// Device/Application/Vizualization/7_inch/_Actuators
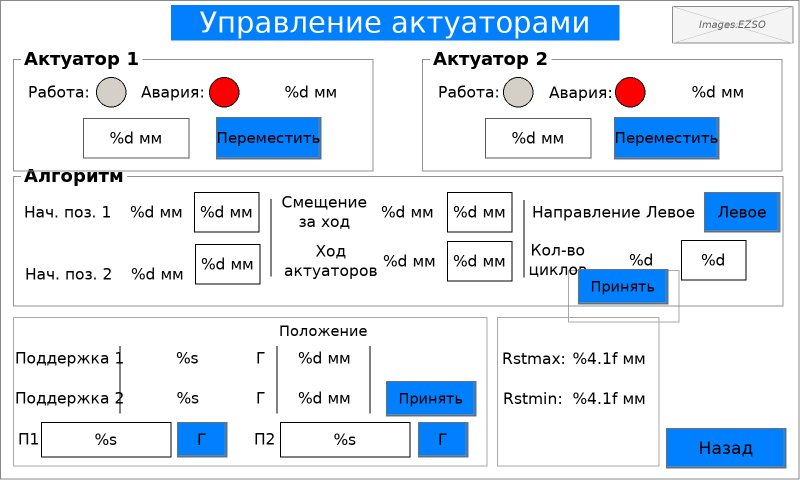
VISUALIZATION _Actuators  // 800x480, background image Images.background
    RoundedRectangle (568,270 111x52)
    GroupBox (13,168 770x138), "Алгоритм"
        Label (507,75 76x34), "Кол-во циклов"
        Label (516,27 113x34), "Направление"
        Button (691,24 76x40), "Левое", text list: 'DirectRotation', text index: setPoint.bDirRotate
            toggle setPoint.bDirRotate
        RoundedRectangle (668,72 65x40), "%d", text variable: setPoint.iCountCycle
            OnMouseClick: write the text variable via VisuDialogs.Numpad, min 0, max 360, title 'Input'
        RoundedRectangle (181,24 65x40), "%d мм", text variable: setPoint.iActuatorsStartPos[0]
            OnMouseClick: write the text variable via VisuDialogs.Numpad, min 0, max SP.iMaxActuatorsMove, title 'Input'
        RoundedRectangle (434,24 65x40), "%d мм", text variable: setPoint.iActuatorsStep
            OnMouseClick: write the text variable via VisuDialogs.Numpad, min 0, max SP.iMaxActuatorsMove, title 'Input'
        Label (8,27 98x34), "Нач. поз. 1"
        Label (260,27 103x34), "Смещение за ход"
        Rectangle (111,29 65x30), "%d мм", text variable: curPoint.iActuatorsStartPos[0]
        Line (258,108) (258,31)
        Line (511,109) (511,32)
        Rectangle (596,77 65x30), "%d", text variable: curPoint.iCountCycle
        Rectangle (362,29 65x30), "%d мм", text variable: curPoint.iActuatorsStep
        Rectangle (625,29 65x30), "Левое", text list: 'DirectRotation', text index: curPoint.bDirRotate
        Button (565,101 90x35), "Принять", pressed state: Global_Variables.btnAccept.bAct
            tap Global_Variables.btnAccept.bAct
        RoundedRectangle (182,76 65x40), "%d мм", text variable: setPoint.iActuatorsStartPos[1]
            OnMouseClick: write the text variable via VisuDialogs.Numpad, min 0, max SP.iMaxActuatorsMove, title 'Input'
        Rectangle (364,78 65x30), "%d мм", text variable: curPoint.iActuatorsMove
        RoundedRectangle (434,73 65x40), "%d мм", text variable: setPoint.iActuatorsMove
            OnMouseClick: write the text variable via VisuDialogs.Numpad, min 0, max SP.iMaxActuatorsMove, title 'Input'
        Label (271,76 94x34), "Ход актуаторов"
    RoundedRectangle (497,317 162x149)
    RoundedRectangle (13,317 474x149)
    Image (672,6 121x37), image: Images.EZSO
    Button (666,428 120x40), "Назад"
        OnMouseDown:  Assign=_MAIN_7inch, Type=Previous
        OnMouseDown: execute { Actuators.bManualMode := FALSE; }
    Rectangle (171,5 448x35), "Управление актуаторами"
    GroupBox (13,51 360x120), "Актуатор 1"
        RoundedRectangle (70,67 106x40), "%d мм", text variable: Actuators.fbAct1.iSetp
            OnMouseClick: write the text variable via VisuDialogs.Numpad, min 0, max SP.rMaxLength, title 'Input'
        Button (203,66 105x42), "Переместить", pressed state: Actuators.fbAct1.bBtnStart
            tap Actuators.fbAct1.bBtnStart
        Rectangle (240,26 116x30), "%d мм", text variable: Actuators.fbAct1.iCurLength
        Label (12,25 68x32), "Работа:"
        Ellipse (83,26 30x30), colour toggle: Actuators.bDr1_enable
        Label (125,25 68x32), "Авария:"
        Ellipse (196,26 30x30), colour toggle: Actuators.bDr2_error
    GroupBox (422,51 360x120), "Актуатор 2"
        RoundedRectangle (63,67 106x40), "%d мм", text variable: Actuators.fbAct2.iSetp
            OnMouseClick: write the text variable via VisuDialogs.Numpad, min 0, max SP.rMaxLength, title 'Input'
        Button (192,66 105x42), "Переместить", pressed state: Actuators.fbAct2.bBtnStart
            tap Actuators.fbAct2.bBtnStart
        Rectangle (238,26 116x30), "%d мм", text variable: Actuators.fbAct2.iCurLength
        Label (13,24 67x34), "Работа:"
        Ellipse (81,26 30x30), colour toggle: Actuators.bDr1_enable
        Label (124,26 68x31), "Авария:"
        Ellipse (193,26 30x30), colour toggle: Actuators.bDr2_error
    Line (120,413) (120,346)
    Line (277,413) (277,346)
    Button (418,422 50x35), "Г", text list: 'TypeSetup', text index: setPoint.support[1].bPosition
        toggle setPoint.support[1].bPosition
    Button (177,422 50x35), "Г", text list: 'TypeSetup', text index: setPoint.support[0].bPosition
        toggle setPoint.support[0].bPosition
    RoundedRectangle (280,422 130x35), "%s", text variable: setPoint.support[1].name
        OnMouseClick:  Dialog=_Diag_supKey, Parameters={stValue: setPoint.support[1]}, Selected={1: }, OpenModal=True, PositionX=300, PositionY=150
    RoundedRectangle (41,422 130x35), "%s", text variable: setPoint.support[0].name
        OnMouseClick:  Dialog=_Diag_supKey, Parameters={stValue: setPoint.support[0]}, Selected={1: }, OpenModal=True, PositionX=300, PositionY=150
    Label (12,381 105x34), "Поддержка 2"
    Label (12,341 105x34), "Поддержка 1"
    Line (370,413) (370,346)
    Label (276,314 96x34), "Положение"
    Rectangle (286,343 77x30), "%d мм", text variable: Actuators.iCurLenSuport1
    Rectangle (286,383 77x30), "%d мм", text variable: Actuators.iCurLenSuport2
    RoundedRectangle (564,341 90x35), "%4.1f мм", text variable: curPoint.rRstmax
    Label (499,343 66x31), "Rstmax:"
    Label (500,383 65x31), "Rstmin:"
    RoundedRectangle (564,381 90x35), "%4.1f мм", text variable: curPoint.rRstmin
    Rectangle (123,343 129x30), "%s", text variable: curPoint.support[0].name
    Rectangle (123,383 130x30), "%s", text variable: curPoint.support[1].name
    Rectangle (246,343 30x30), "Г", text list: 'TypeSetup', text index: curPoint.support[0].bPosition
    Rectangle (246,383 30x30), "Г", text list: 'TypeSetup', text index: curPoint.support[1].bPosition
    Button (386,381 90x35), "Принять", pressed state: Global_Variables.btnAccept.bSup
        tap Global_Variables.btnAccept.bSup
    Label (15,426 31x26), "П1"
    Label (251,426 31x26), "П2"
    Label (22,257 98x34), "Нач. поз. 2"
    Rectangle (125,259 65x30), "%d мм", text variable: curPoint.iActuatorsStartPos[1]
END_VISUALIZATION

// Device/Application/Vizualization/7_inch/_SettingsEquipment
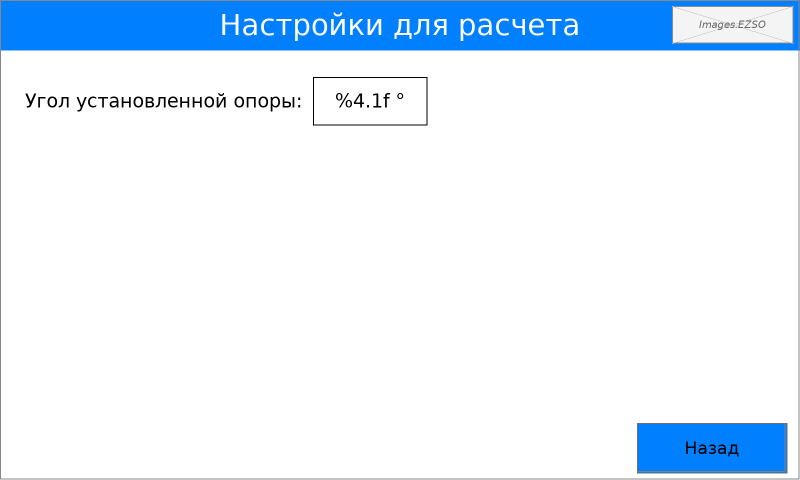
VISUALIZATION _SettingsEquipment  // 800x480
    Rectangle (0,0 800x50), "Настройки для расчета"
    Image (672,6 121x37), image: Images.EZSO
    Button (637,423 150x50), "Назад"
        OnMouseDown:  Assign=_MAIN_7inch, Type=Previous
    RoundedRectangle (313,77 114x48), "%4.1f °", text variable: SP.rInitAngleSupport
        OnValueChanged: execute { CalcTech.rAngle_support:=sp.rInitAngleSupport; }
        OnMouseClick: write the text variable via VisuDialogs.Numpad, min 0, max 359
    Label (22,80 295x42), "Угол установленной опоры:"
END_VISUALIZATION

// Device/Application/Vizualization/7_inch/_Diag_geomtry_rec
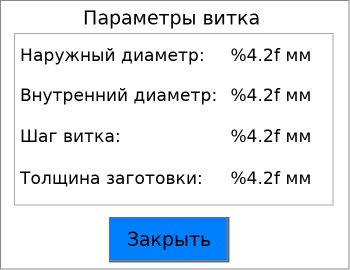
VISUALIZATION _Diag_geomtry_rec  // 350x270
    Button (109,217 120x45), "Закрыть"
        toggle bGoCalc
        OnMouseClick:  Dialog=Current Dialog, Result=OK, NumpadKeypadSet=True
    RoundedRectangle (214,71 114x48), "%4.2f мм", text variable: recipes.Screw.rInner_diam
    Label (17,74 223x42), "Внутренний диаметр:"
    RoundedRectangle (214,31 114x48), "%4.2f мм", text variable: recipes.Screw.rOut_diam
        OnMouseClick: write the text variable via VisuDialogs.Numpad
    Label (17,34 223x42), "Наружный диаметр:"
    RoundedRectangle (214,112 114x48), "%4.2f мм", text variable: recipes.Screw.rTurn_step
    Label (17,115 223x42), "Шаг витка:"
    RoundedRectangle (214,154 114x48), "%4.2f мм", text variable: recipes.Screw.rWidth
    Label (17,157 223x42), "Толщина заготовки:"
    Label (80,1 185x34), "Параметры витка"
    RoundedRectangle (14,33 319x172)
END_VISUALIZATION

// Device/Application/Vizualization/7_inch/_Support
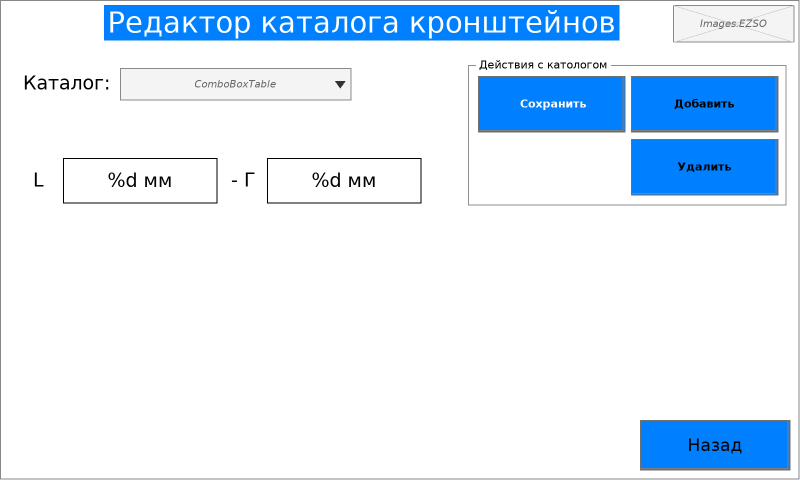
VISUALIZATION _Support  // 800x480, background image Images.background
    GroupBox (468,57 318x148), "Действия с катологом"
        Button (163,82 147x56), "Удалить"
            OnMouseClick: execute { recipes.DelData(3); }
        Button (163,19 147x56), "Добавить"
            OnMouseClick: execute { recipes.addData(3); }
        Button (10,19 147x56), "Сохранить"
            OnMouseClick: execute { recipes.setData(3); }
    Label (30,165 31x30), "L"
    Label (20,68 99x30), "Каталог:"
    Image (673,5 121x37), image: Images.EZSO
    Rectangle (104,5 515x35), "Редактор каталога кронштейнов"
    Button (640,420 150x50), "Назад"
        OnMouseDown:  Assign=_Equipment, Type=Assignment
        OnMouseDown:  ExecuteCommand=ExecuteCommand=[Command=ReadRecipe, Value=sRecGroupName3, Value2=sRecName3]
    ComboBoxTable (120,68 231x32), variable: recipes.idxArSupport, data array: arSupports
        p1014161805: Global_Variables.SIZE_SUPPORT - 0 + 1
        p338671338: arrSteel_buf[INDEX].G
        p2170511999: arrSteel_buf[INDEX].t
        p3854506369: arSupports[INDEX].arLength
        p1892666644: arSupports[INDEX].name
        OnValueChanged: execute { recipes.GetData(3); }
    RoundedRectangle (63,158 154x45), "%d мм", text variable: recipes.Support.arLength[0]
        OnMouseClick: write the text variable via VisuDialogs.Numpad, min -999, max 999, title 'Input'
    RoundedRectangle (267,158 154x45), "%d мм", text variable: recipes.Support.arLength[1]
        OnMouseClick: write the text variable via VisuDialogs.Numpad, min -999, max 999, title 'Input'
    Label (228,165 31x30), "- Г"
END_VISUALIZATION

// Device/Application/Vizualization/7_inch/_Equipment_2
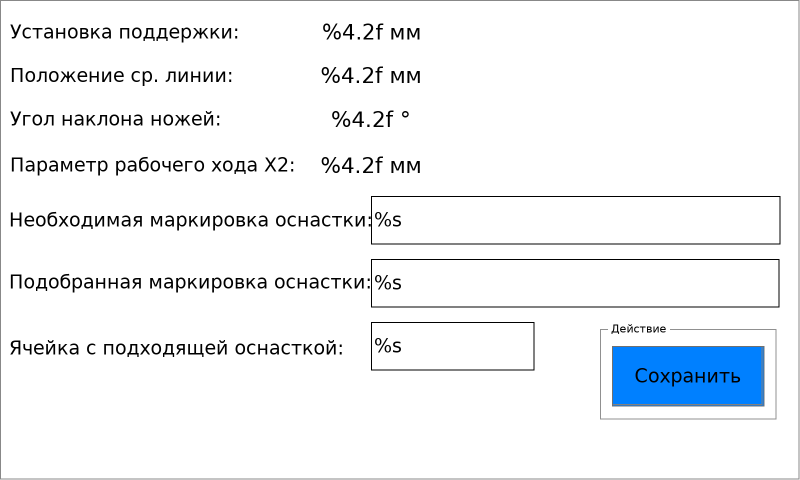
VISUALIZATION _Equipment_2  // 800x480
    Label (6,327 338x42), "Ячейка с подходящей оснасткой:"
    Label (6,198 396x44), "Необходимая маркировка оснастки:"
    RoundedRectangle (371,196 409x48), "%s", text variable: CalcTech.msEquipment.bestFind.name
    Label (7,55 231x41), "Положение ср. линии:"
    Label (7,15 232x34), "Установка поддержки:"
    RoundedRectangle (371,259 408x48), "%s", text variable: CalcTech.msEquipment.find.name
    Label (7,98 223x42), "Угол наклона ножей:"
    Label (7,144 322x42), "Параметр рабочего хода Х2:"
    Label (6,261 360x42), "Подобранная маркировка оснастки:"
    Rectangle (322,17 100x30), "%4.2f мм", text variable: CalcTech.rMsFactInstal_support
    Rectangle (320,62 102x27), "%4.2f мм", text variable: CalcTech.rMsFactMidle_line
    Rectangle (320,152 102x27), "%4.2f мм", text variable: CalcTech.rMsX2
    Rectangle (320,106 102x27), "%4.2f °", text variable: CalcTech.rMsAngle_knives
    RoundedRectangle (371,322 163x48), "%s", text variable: CalcTech.msEquipment.find.place
    GroupBox (600,321 176x98), "Действие"
        Button (12,25 152x60), "Сохранить"
            OnMouseClick:  Dialog=_Diag_save, PositionX=300, PositionY=150
END_VISUALIZATION

// Device/Application/Vizualization/7_inch/_Equipment_3
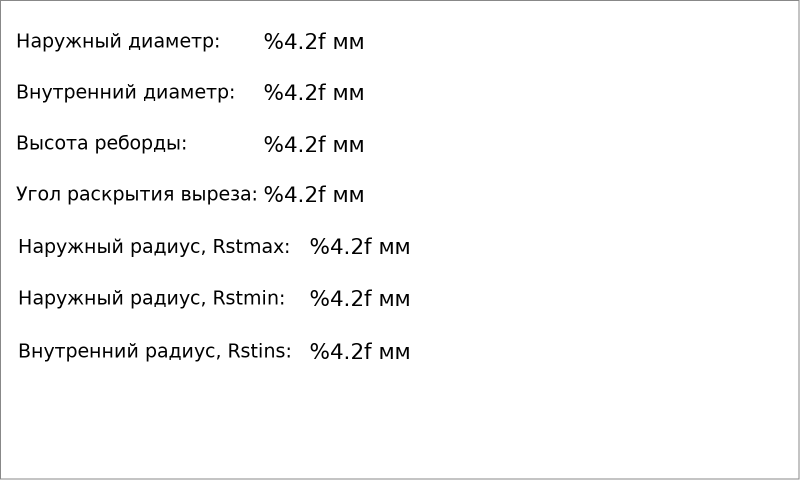
VISUALIZATION _Equipment_3  // 800x480
    Label (13,71 223x42), "Внутренний диаметр:"
    Label (13,20 223x42), "Наружный диаметр:"
    Label (13,122 223x42), "Высота реборды:"
    Label (13,173 250x42), "Угол раскрытия выреза:"
    Rectangle (263,181 102x27), "%4.2f мм", text variable: CalcTech.rWpAngle
    Rectangle (263,79 102x27), "%4.2f мм", text variable: CalcTech.rWpInner_diam
    Rectangle (263,28 102x27), "%4.2f мм", text variable: CalcTech.rWpOut_diam
    Rectangle (263,131 102x27), "%4.2f мм", text variable: CalcTech.rWpRebordHeight
    Label (15,224 290x45), "Наружный радиус, Rstmax:", invisible if: not CalcTech.bEnConicalScrew
    Rectangle (309,234 102x25), "%4.2f мм", text variable: CalcTech.rRstmax, invisible if: not CalcTech.bEnConicalScrew
    Label (15,278 290x40), "Наружный радиус, Rstmin:", invisible if: not CalcTech.bEnConicalScrew
    Label (15,331 289x40), "Внутренний радиус, Rstins:", invisible if: not CalcTech.bEnConicalScrew
    Rectangle (309,286 102x25), "%4.2f мм", text variable: CalcTech.rRstmin, invisible if: not CalcTech.bEnConicalScrew
    Rectangle (309,339 102x25), "%4.2f мм", text variable: CalcTech.rRstins, invisible if: not CalcTech.bEnConicalScrew
END_VISUALIZATION

// Device/Application/Vizualization/7_inch/_Diag_WARNING
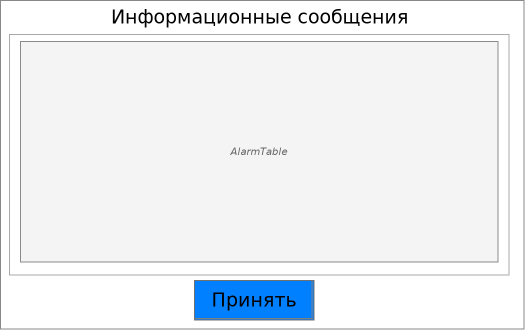
VISUALIZATION _Diag_WARNING  // 525x330
VAR_IN_OUT
	stValue:WSTRING;	
END_VAR
VAR
	sDirection: INT;
	sTypeEquip:	INT;
	sHeight: WSTRING;
	sAngle:	WSTRING;
	sMidle:	WSTRING;	
END_VAR
    RoundedRectangle (9,34 500x241)
    Button (194,280 120x40), "Принять"
        tap bReset
        OnMouseDown:  Dialog=Current Dialog, Result=OK, NumpadKeypadSet=True
    AlarmTable (20,41 478x221)
        p1521930926: WarningGroup
        p1663851261: Warning
    Label (108,0 308x34), "Информационные сообщения"
END_VISUALIZATION

// Device/Application/Vizualization/7_inch/_TypeMachine
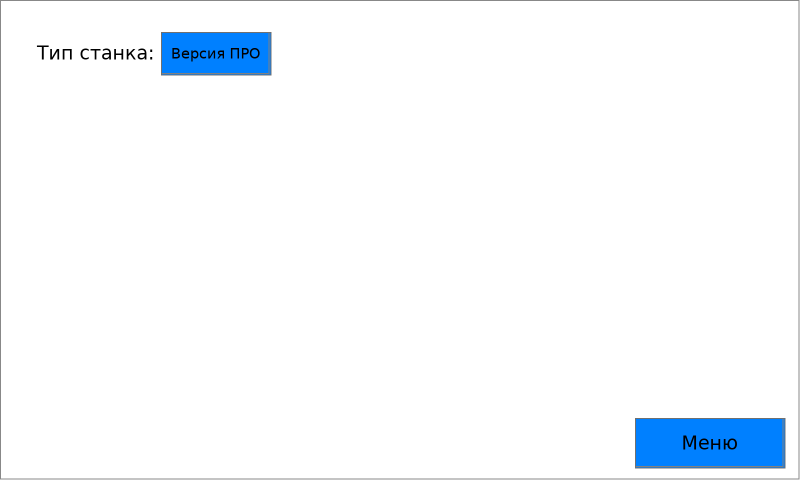
VISUALIZATION _TypeMachine  // 800x480
    Button (161,32 110x43), "Версия ПРО", colour toggle: SP.bEnAutoMatrix
        toggle SP.bEnAutoMatrix
    Label (34,32 129x42), "Тип станка:"
    Button (635,418 150x50), "Меню"
        OnMouseDown:  Assign=_SettingsMain_7inch, Type=Assignment
END_VISUALIZATION

// Device/Application/Vizualization/7_inch/_Diag_support_rec
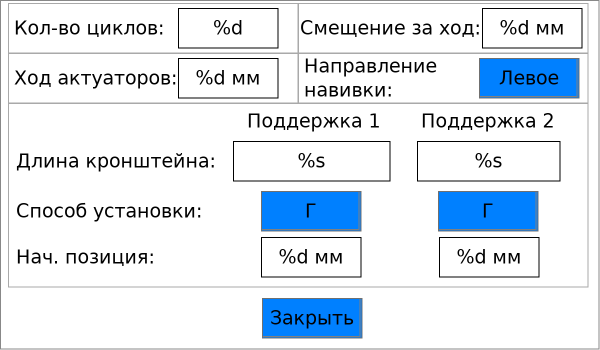
VISUALIZATION _Diag_support_rec  // 600x350
    RoundedRectangle (298,53 290x50)
    RoundedRectangle (8,3 290x50)
    RoundedRectangle (8,53 290x50)
    RoundedRectangle (298,3 290x50)
    RoundedRectangle (8,103 580x184)
    Button (262,298 100x40), "Закрыть"
        toggle bGoCalc
        OnMouseClick:  Dialog=Current Dialog, Result=OK, NumpadKeypadSet=True
    Label (11,11 153x34), "Кол-во циклов:"
    Label (11,61 168x34), "Ход актуаторов:"
    Label (297,11 191x34), "Смещение за ход:"
    Label (13,240 147x34), "Нач. позиция:"
    Label (244,104 134x34), "Поддержка 1"
    Label (13,144 204x34), "Длина кронштейна:"
    Label (13,194 194x34), "Способ установки:"
    Label (418,104 140x34), "Поддержка 2"
    Label (301,57 156x42), "Направление навивки:"
    Button (479,58 100x40), "Левое", text list: 'DirectRotation', text index: recipes.Screw.bDirRotate
        toggle recipes.Screw.bDirRotate
    RoundedRectangle (178,8 100x40), "%d", text variable: recipes.Screw.iCountCycle
        OnMouseClick: write the text variable via VisuDialogs.Numpad, min 0, max 360, title 'Input'
    RoundedRectangle (178,58 100x40), "%d мм", text variable: recipes.Screw.iActuatorsMove
        OnMouseClick: write the text variable via VisuDialogs.Numpad, min 0, max SP.iMaxActuatorsMove, title 'Input'
    RoundedRectangle (482,8 100x40), "%d мм", text variable: recipes.Screw.iActuatorsStep
        OnMouseClick: write the text variable via VisuDialogs.Numpad, min 0, max SP.iMaxActuatorsMove, title 'Input'
    RoundedRectangle (261,237 100x40), "%d мм", text variable: recipes.Screw.iActuatorsStartPos[0]
        OnMouseClick: write the text variable via VisuDialogs.Numpad, min 0, max SP.iMaxActuatorsMove, title 'Input'
    RoundedRectangle (233,141 157x40), "%s", text variable: recipes.Screw.support[0].name
        OnMouseClick:  Dialog=_Diag_supKey, Parameters={stValue: recipes.Screw.support[0]}, Selected={6: , 1: }, OpenModal=True, PositionX=300, PositionY=150
    RoundedRectangle (417,141 143x40), "%s", text variable: recipes.Screw.support[1].name
        OnMouseClick:  Dialog=_Diag_supKey, Parameters={stValue: recipes.Screw.support[1]}, Selected={6: , 1: }, OpenModal=True, PositionX=300, PositionY=150
    Button (261,191 100x40), "Г", text list: 'TypeSetup', text index: recipes.Screw.support[0].bPosition
        toggle recipes.Screw.support[0].bPosition
    Button (438,191 100x40), "Г", text list: 'TypeSetup', text index: recipes.Screw.support[1].bPosition
        toggle recipes.Screw.support[1].bPosition
    RoundedRectangle (439,237 100x40), "%d мм", text variable: recipes.Screw.iActuatorsStartPos[1]
        OnMouseClick: write the text variable via VisuDialogs.Numpad, min 0, max SP.iMaxActuatorsMove, title 'Input'
END_VISUALIZATION

// Device/Application/Vizualization/7_inch/_Equip_7inch
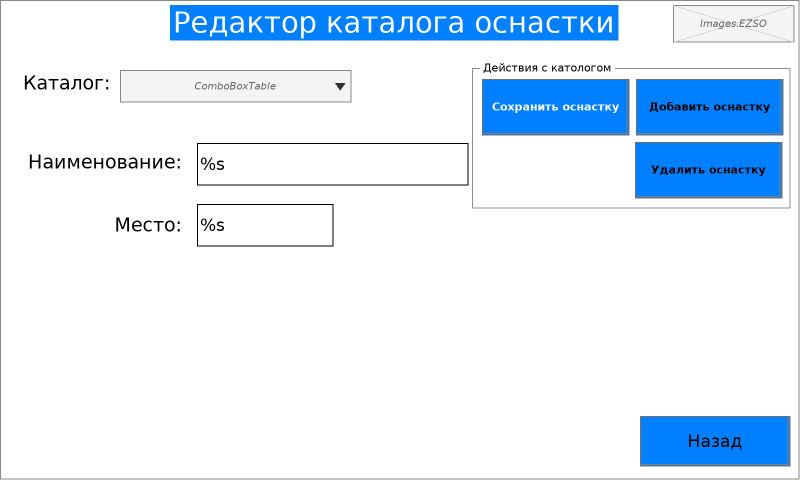
VISUALIZATION _Equip_7inch  // 800x480, background image Images.background
    Label (20,68 99x30), "Каталог:"
    Image (673,5 121x37), image: Images.EZSO
    RoundedRectangle (197,143 271x42), "%s", text variable: recipes.Equip.name
        OnMouseDown:  Dialog=_Diag_equip, Parameters={sHeight: , stValue: recipes.Equip.name, sTypeEquip: , sMidle: , sDirection: , sAngle: }, Selected={1: }, OpenModal=True, PositionX=100, PositionY=120
    RoundedRectangle (197,204 136x42), "%s", text variable: recipes.Equip.place
        OnMouseClick: write the text variable via VisuDialogs.Numpad, title 'Input'
    Label (109,210 76x30), "Место:"
    GroupBox (472,60 318x148), "Действия с катологом"
        Button (163,82 147x56), "Удалить оснастку"
            OnMouseClick: execute { recipes.DelData(1); }
        Button (164,19 147x56), "Добавить оснастку"
            OnMouseClick: execute { recipes.addData(1); }
        Button (10,19 147x56), "Сохранить оснастку"
            OnMouseClick: execute { recipes.setData(1); }
    Label (11,147 174x30), "Наименование:"
    Rectangle (170,5 448x35), "Редактор каталога оснастки"
    Button (640,416 150x50), "Назад"
        OnMouseDown:  Assign=_Equipment, Type=Assignment
        OnMouseDown:  ExecuteCommand=ExecuteCommand=[Command=ReadRecipe, Value=sRecGroupName2, Value2=sRecName2]
    ComboBoxTable (120,70 231x32), variable: recipes.idxArEquip, data array: ArEquip
        p1014161805: Global_Variables.SIZE_EQUIPS - 0 + 1
        p338671338: arrEquip_buf[INDEX].access
        p2170511999: arrSteel_buf[INDEX].t
        p3854506369: ArEquip[INDEX].place
        p1892666644: ArEquip[INDEX].name
        OnValueChanged: execute { recipes.getData(1); }
END_VISUALIZATION

// Device/Application/Vizualization/7_inch/_Equipment_4
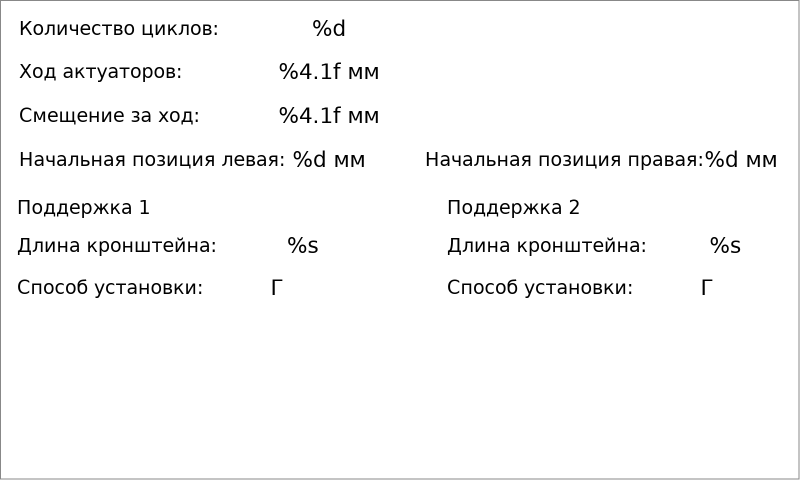
VISUALIZATION _Equipment_4  // 800x480
    Label (16,6 227x45), "Количество циклов:"
    Rectangle (278,16 102x25), "%d", text variable: CalcTech.iCountCycle
    Label (16,49 227x45), "Ход актуаторов:"
    Rectangle (278,59 102x25), "%4.1f мм", text variable: CalcTech.rActuatorsMove
    Label (16,93 227x45), "Смещение за ход:"
    Rectangle (278,103 102x25), "%4.1f мм", text variable: CalcTech.rActuatorsStep
    Label (16,137 274x45), "Начальная позиция левая:"
    Rectangle (278,147 102x25), "%d мм", text variable: CalcTech.iStartSupPos[0]
    Label (14,185 227x45), "Поддержка 1"
    Rectangle (226,233 154x25), "%s", text variable: CalcTech.support[0].name
    Label (14,223 227x45), "Длина кронштейна:"
    Rectangle (238,275 78x25), "Г", text list: 'TypeSetup', text index: CalcTech.support[0].bPosition
    Label (14,265 227x45), "Способ установки:"
    Label (444,185 227x45), "Поддержка 2"
    Rectangle (656,233 139x25), "%s", text variable: CalcTech.support[1].name
    Label (444,223 227x45), "Длина кронштейна:"
    Rectangle (668,275 78x25), "Г", text list: 'TypeSetup', text index: CalcTech.support[1].bPosition
    Label (444,265 227x45), "Способ установки:"
    Label (422,137 280x45), "Начальная позиция правая:"
    Rectangle (690,147 102x25), "%d мм", text variable: CalcTech.iStartSupPos[1]
END_VISUALIZATION

// Device/Application/Vizualization/7_inch/_Diag_save
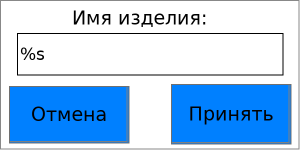
VISUALIZATION _Diag_save  // 300x150
    Button (171,84 120x60), "Принять"
        OnMouseClick: execute { recipes.screw := calcTech.dataForRec; recipes.AddData(0); }
        OnMouseClick:  Dialog=Current Dialog, Result=OK, NumpadKeypadSet=True
        OnMouseClick:  Assign=_Recipe_7inch, Type=Assignment
    Button (9,86 120x57), "Отмена"
        OnMouseClick:  Dialog=_Diag_save, Result=None, NumpadKeypadSet=True
    Label (69,1 143x34), "Имя изделия:"
    RoundedRectangle (17,33 266x42), "%s", text variable: CalcTech.dataForRec.name
        OnMouseClick: write the text variable via VisuKbEnRu.Keypad, max 20, title 'Input'
END_VISUALIZATION

// Device/Application/Vizualization/7_inch/_Equipment_1
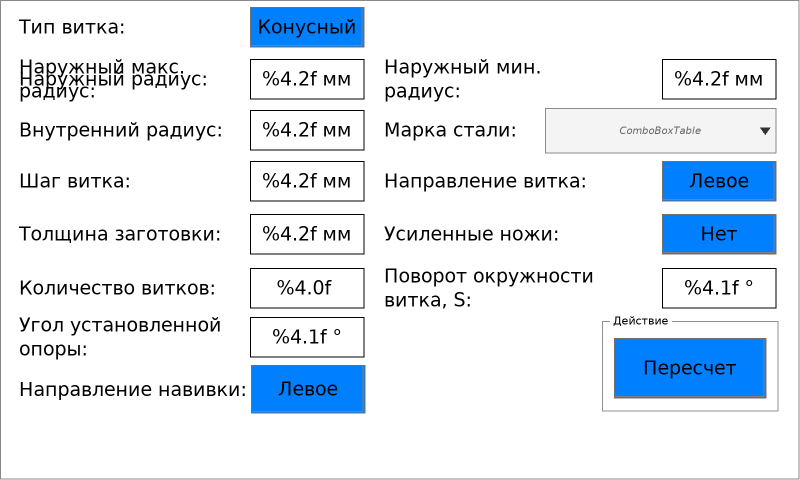
VISUALIZATION _Equipment_1  // 800x480
    RoundedRectangle (250,317 114x40), "%4.1f °", text variable: CalcTech.rAngle_support
        OnMouseClick: write the text variable via VisuDialogs.Numpad, min 0, max 360
    Label (16,316 219x42), "Угол установленной опоры:"
    Label (16,266 223x44), "Количество витков:"
    RoundedRectangle (250,268 114x40), "%4.0f", text variable: CalcTech.rCount_turn
        OnMouseClick: write the text variable via VisuDialogs.Numpad, min 0, max 1000
    RoundedRectangle (250,110 114x40), "%4.2f мм", text variable: CalcTech.rRins
        OnMouseClick: write the text variable via VisuDialogs.Numpad, min 0, max 1000
    Label (16,109 223x42), "Внутренний радиус:"
    RoundedRectangle (250,59 114x40), "%4.2f мм", text variable: CalcTech.rRoutmax
        OnMouseClick: write the text variable via VisuDialogs.Numpad, min 0, max 1000
    Label (16,58 223x42), "Наружный радиус:", invisible if: CalcTech.bEnConicalScrew
    RoundedRectangle (250,161 114x40), "%4.2f мм", text variable: CalcTech.rTurn_step
        OnMouseClick: write the text variable via VisuDialogs.Numpad, min 0, max 1000
    Label (16,160 223x42), "Шаг витка:"
    RoundedRectangle (250,214 114x40), "%4.2f мм", text variable: CalcTech.rWidth
        OnMouseClick: write the text variable via VisuDialogs.Numpad, min 0, max 1000
    Label (16,213 223x42), "Толщина заготовки:"
    Label (381,109 295x42), "Марка стали:"
    Label (381,213 295x42), "Усиленные ножи:"
    Label (381,160 295x42), "Направление витка:"
    Button (662,161 114x40), "Левое", text list: 'Direction', text index: CalcTech.bDirection
        toggle CalcTech.bDirection
    Button (662,214 114x40), "Нет", pressed state: CalcTech.bStrengthened, text list: 'NoYes', text index: CalcTech.bStrengthened
        toggle CalcTech.bStrengthened
    ComboBoxTable (545,108 231x45), variable: recipes.idxArSteel, data array: arSteel
        p1014161805: Global_Variables.SIZE_STEELS - 0 + 1
        p3854506369: arSteel[INDEX].name
        p1892666644: arSteel[INDEX].density
        p338671338: arSteel[INDEX].G
        p2170511999: arSteel[INDEX].t
        p1755163831: arrSteel_buf[INDEX].G
        p4092479075: arrSteel_buf[INDEX].t
        OnValueChanged: execute { CalcTech.steel := arSteel[recipes.idxArSteel]; }
    GroupBox (602,313 176x98), "Действие"
        Button (12,25 152x60), "Пересчет"
            tap bGoCalc
    RoundedRectangle (662,59 114x40), "%4.2f мм", text variable: CalcTech.rRoutmin, invisible if: not CalcTech.bEnConicalScrew
        OnMouseClick: write the text variable via VisuDialogs.Numpad, min 0, max 1000
    Label (381,58 171x42), "Наружный мин. радиус:", invisible if: not CalcTech.bEnConicalScrew
    RoundedRectangle (662,268 114x40), "%4.1f °", text variable: CalcTech.rRotationCircle, invisible if: not CalcTech.bEnConicalScrew
        OnMouseClick: write the text variable via VisuDialogs.Numpad, min 0, max 360
    Label (381,267 219x42), "Поворот окружности витка, S:", invisible if: not CalcTech.bEnConicalScrew
    Label (16,58 266x42), "Наружный макс. радиус:", invisible if: not CalcTech.bEnConicalScrew
    Label (16,6 114x42), "Тип витка:", invisible if: NOT SP.bEnAutoMatrix
    Button (250,7 114x40), "Конусный", colour toggle: CalcTech.bEnConicalScrew, invisible if: NOT SP.bEnAutoMatrix
        toggle CalcTech.bEnConicalScrew
    Label (16,370 233x39), "Направление навивки:"
    Button (251,365 114x48), "Левое", text list: 'DirectRotation', text index: CalcTech.bDirRotation
        toggle CalcTech.bDirection
END_VISUALIZATION

// Device/Application/Vizualization/7_inch/_Diag_geomtry_work
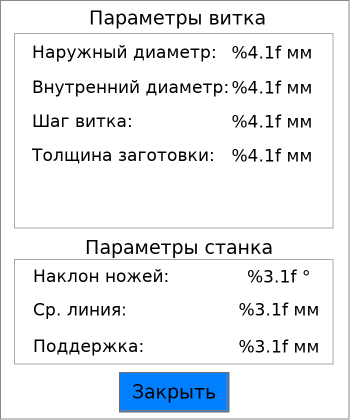
VISUALIZATION _Diag_geomtry_work  // 350x420
    RoundedRectangle (14,33 319x195)
    RoundedRectangle (14,259 319x105)
    Rectangle (224,292 110x35), "%3.1f мм", text variable: curPoint.rMidle_line
    Label (82,232 199x31), "Параметры станка"
    Button (119,372 110x40), "Закрыть"
        toggle bGoCalc
        OnMouseClick:  Dialog=Current Dialog, Result=None, NumpadKeypadSet=True
    RoundedRectangle (217,70 110x35), "%4.1f мм", text variable: curPoint.rInner_diam
    Label (29,66 186x42), "Внутренний диаметр:"
    RoundedRectangle (217,35 110x35), "%4.1f мм", text variable: curPoint.rOut_diam
    Label (29,31 179x42), "Наружный диаметр:"
    RoundedRectangle (217,104 110x35), "%4.1f мм", text variable: curPoint.rTurn_step
    Label (29,100 101x42), "Шаг витка:"
    Rectangle (217,138 110x35), "%4.1f мм", text variable: curPoint.rWidth
    Label (29,134 176x42), "Толщина заготовки:"
    Rectangle (224,329 110x35), "%3.1f мм", text variable: curPoint.rInstal_support
    Rectangle (224,259 110x35), "%3.1f °", text variable: curPoint.rAngle_knives
    Label (30,289 95x41), "Ср. линия:"
    Label (30,329 109x34), "Поддержка:"
    Label (30,255 136x42), "Наклон ножей:"
    Label (86,1 185x34), "Параметры витка"
END_VISUALIZATION

// Device/Application/Vizualization/7_inch/_Steel_7inch
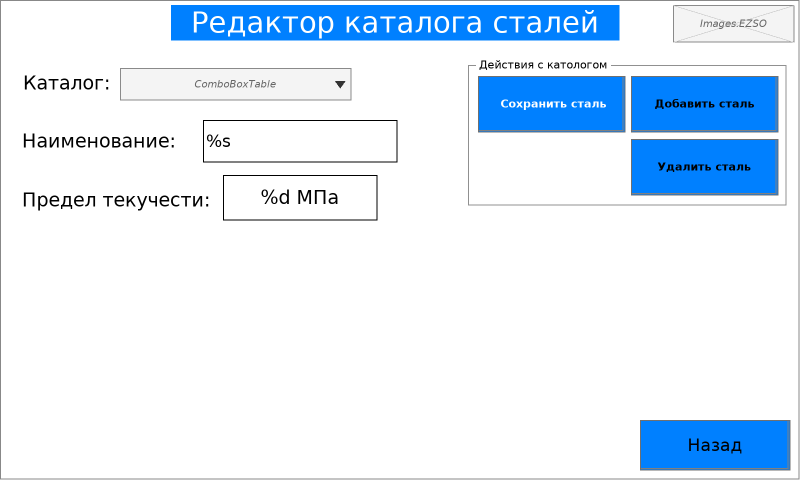
VISUALIZATION _Steel_7inch  // 800x480, background image Images.background
    GroupBox (468,57 318x148), "Действия с катологом"
        Button (163,82 147x56), "Удалить сталь"
            OnMouseClick: execute { recipes.DelData(2); }
        Button (163,19 147x56), "Добавить сталь"
            OnMouseClick: execute { recipes.addData(2); }
        Button (10,19 147x56), "Сохранить сталь"
            OnMouseClick: execute { recipes.SetData(2); }
    Label (19,185 200x30), "Предел текучести:"
    Label (19,126 174x30), "Наименование:"
    Label (20,68 99x30), "Каталог:"
    Image (673,5 121x37), image: Images.EZSO
    Rectangle (171,5 448x35), "Редактор каталога сталей"
    Button (640,420 150x50), "Назад"
        OnMouseDown:  Assign=_Equipment, Type=Assignment
        OnMouseDown:  ExecuteCommand=ExecuteCommand=[Command=ReadRecipe, Value=sRecGroupName1, Value2=sRecName1]
    ComboBoxTable (120,68 231x32), variable: recipes.idxArSteel, data array: ArSteel
        p1014161805: Global_Variables.SIZE_STEELS - 0 + 1
        p338671338: arrSteel_buf[INDEX].G
        p2170511999: arrSteel_buf[INDEX].t
        p3854506369: ArSteel[INDEX].t
        p1892666644: ArSteel[INDEX].name
        OnValueChanged: execute { recipes.getData(2); }
    RoundedRectangle (223,175 154x45), "%d МПа", text variable: recipes.Steel.t
        OnMouseClick: write the text variable via VisuDialogs.Numpad, min 0, max 999999, title 'Input'
    RoundedRectangle (203,120 194x42), "%s", text variable: recipes.Steel.name
        OnMouseClick: write the text variable via VisuKbEnRu.Keypad, title 'Input'
END_VISUALIZATION

// Device/Application/Vizualization/7_inch/_SettingsSens_7inch
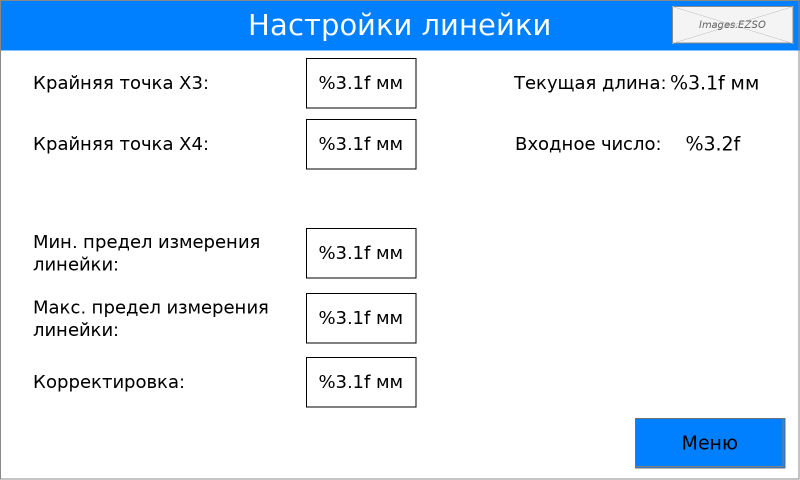
VISUALIZATION _SettingsSens_7inch  // 800x480
    Button (635,418 150x50), "Меню"
        OnMouseDown:  Assign=_SettingsMain_7inch, Type=Assignment
    RoundedRectangle (306,357 110x50), "%3.1f мм", text variable: SP.rOffset
        OnMouseClick: write the text variable via VisuDialogs.Numpad, min -999, max 999, title 'Input'
    RoundedRectangle (306,58 110x50), "%3.1f мм", text variable: SP.rMinPoint
        OnMouseClick: write the text variable via VisuDialogs.Numpad, min -999, max 999, title 'Input'
    RoundedRectangle (306,119 110x50), "%3.1f мм", text variable: SP.rMaxPoint
        OnMouseClick: write the text variable via VisuDialogs.Numpad, min -999, max 999, title 'Input'
    Label (30,367 190x30), "Корректировка:"
    Label (30,63 209x40), "Крайняя точка Х3:"
    Label (30,122 244x44), "Крайняя точка Х4:"
    Rectangle (0,0 800x50), "Настройки линейки"
    Label (30,233 247x40), "Мин. предел измерения линейки:"
    Label (30,290 257x57), "Макс. предел измерения линейки:"
    RoundedRectangle (306,228 110x50), "%3.1f мм", text variable: SP.rMinLength
        OnMouseClick: write the text variable via VisuDialogs.Numpad, min -999, max 999, title 'Input'
    RoundedRectangle (306,293 110x50), "%3.1f мм", text variable: SP.rMaxLength
        OnMouseClick: write the text variable via VisuDialogs.Numpad, min -999, max 9999, title 'Input'
    Image (672,6 121x37), image: Images.EZSO
    Rectangle (665,68 100x30), "%3.1f мм", text variable: Main.snsLenght.rVal
    Label (511,63 159x40), "Текущая длина:"
    Rectangle (666,129 100x30), "%3.2f", text variable: Main.AI_val.rVal
    Label (512,124 153x40), "Входное число:"
END_VISUALIZATION

// Device/Application/Vizualization/Waiting
VISUALIZATION Waiting  // 800x480
    InvisibleInput (10,13 768x448)
        tap Visu_var.exitWait
        OnMouseClick:  Type=Previous
END_VISUALIZATION

// Device/Application/Vizualization/7_inch/_Alarms_7inch
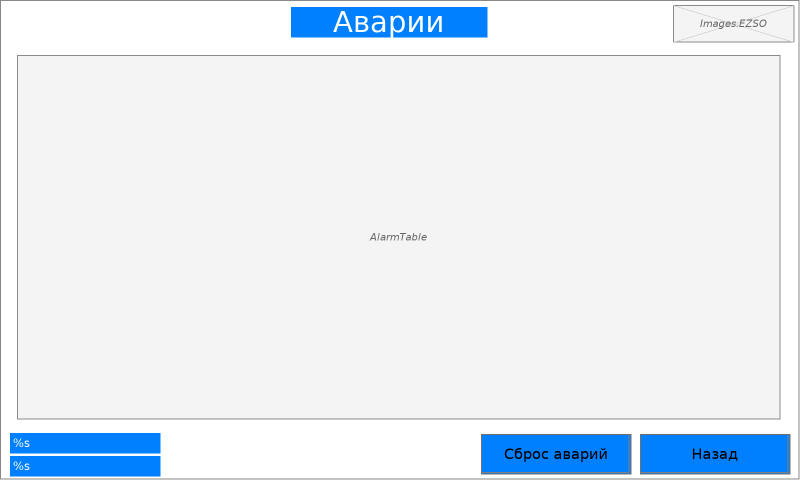
VISUALIZATION _Alarms_7inch  // 800x480, background image Images.background
VAR_IN_OUT
END_VAR
VAR
	bAckSel : BOOL;
	bAckVisible : BOOL;
	bHistory : BOOL;
	bFreezeScrlPos : BOOL;
	sHistoryButtonText :WSTRING := "История аварий";
END_VAR
    Rectangle (10,456 150x20), "%s", text variable: TimeSetup.w_str_dateM
    Rectangle (10,433 150x20), "%s", text variable: TimeSetup.w_str_time
    Button (640,434 150x40), "Назад"
        OnMouseDown:  Assign=_MAIN_Vizu, Type=Previous
    Button (481,434 150x40), "Сброс аварий"
        tap bReset
    AlarmTable (17,55 763x364)
        Column[0]: ColumnTitle=Сообщение
        Column[1]: ColumnTitle=Время
        p1521930926: __All
        p1663851261: __All
        p3266827225: bHistory
    Rectangle (291,7 196x30), "Аварии"
    Image (673,5 121x37), image: Images.EZSO
END_VISUALIZATION

// Device/Application/Vizualization/7_inch/_MAIN_7inch
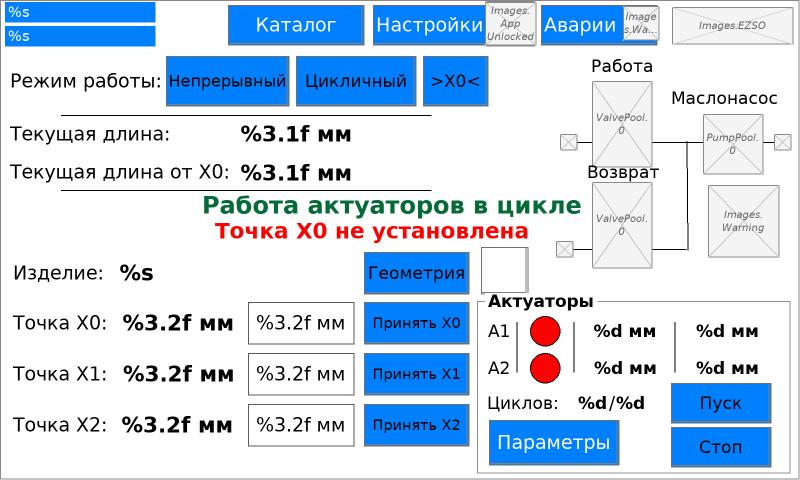
VISUALIZATION _MAIN_7inch  // 800x480, background image Images.background
    Line (652,249) (686,249)
    Line (568,249) (602,249)
    Line (568,142) (602,142)
    Image (560,134 17x16), angle 2, image: Images.Arrow_Black_Left
    Image (556,241 17x16), angle 2, image: Images.Arrow_Black_Left
    Line (629,142) (745,142)
    Line (733,142) (781,142)
    Button (373,5 160x40), "Настройки"
        OnMouseDown:  Assign=_SettingsMain_7inch, Type=Assignment
    Rectangle (5,26 150x20), "%s", text variable: TimeSetup.w_str_dateM
    Rectangle (5,2 150x20), "%s", text variable: TimeSetup.w_str_time
    Button (541,5 116x40), "Аварии", colour toggle: Main.bErrLamp
        OnMouseDown:  Assign=_Alarms_7inch, Type=Assignment
    Image (708,185 71x72), invisible if: NOT Main.bErrLamp OR Main.bSnsH OR Main.bSnsL, image: Images.Warning
    Image (485,1 50x45), invisible if: bLogin, image: Images.AppLocked
        OnMouseClick:  Type=Login
    Image (485,2 51x43), invisible if: not bLogin, image: Images.AppUnlocked
        OnMouseClick:  Type=Logout
    RoundedRectangle (248,302 106x42), "%3.2f мм", text variable: setPoint.rPosX0, invisible if: iMode = 2
        OnMouseClick: write the text variable via VisuDialogs.Numpad, min 0, max SP.rMaxLength, title 'Input'
    Label (10,308 131x30), "Точка X0:"
    Rectangle (231,119 131x30), "%3.1f мм", text variable: Main.snsLenght.rVal
    Label (10,359 131x30), "Точка X1:"
    Label (10,410 131x30), "Точка X2:"
    RoundedRectangle (248,353 106x42), "%3.2f мм", text variable: setPoint.rPosX1, invisible if: iMode = 2
        OnMouseClick: write the text variable via VisuDialogs.Numpad, min 0, max SP.rMaxLength, title 'Input'
    RoundedRectangle (248,404 106x42), "%3.2f мм", text variable: setPoint.rPosX2, invisible if: iMode = 2
        OnMouseClick: write the text variable via VisuDialogs.Numpad, min 0, max SP.rMaxLength, title 'Input'
    Label (7,119 171x30), "Текущая длина:"
    Label (7,157 229x30), "Текущая длина от X0:"
    Rectangle (231,158 131x30), "%3.1f мм", text variable: Main.fbControl.rLengthFromX0
    Image (703,114 60x60), image: PumpPool.0
        p84334746: Visu_var.stMotor
    Image (592,81 60x86), image: ValvePool.0
        p84334746: Visu_var.stValveFrd
    Image (592,182 60x86), image: ValvePool.0
        p84334746: Visu_var.stValveRev
    Line (688,250) (687,141)
    Image (774,134 17x16), angle 2, image: Arrow_Black_Left
    Label (588,51 83x30), "Работа"
    Label (584,157 104x30), "Возврат"
    Label (668,83 131x30), "Маслонасос"
    Image (672,7 121x37), image: Images.EZSO
    Button (364,302 105x42), "Принять Х0", pressed state: Global_Variables.btnAccept.bX0, invisible if: iMode = 2
        tap Global_Variables.btnAccept.bX0
    Button (166,56 123x50), "Непрерывный", colour toggle: iMode = 0
        OnMouseClick: execute { iMode := 0; }
    Button (423,56 65x50), ">X0<", colour toggle: iMode = 2
        OnMouseClick: execute { iMode := 2; }
    Label (7,66 168x30), "Режим работы:"
    Button (296,56 120x50), "Цикличный", colour toggle: iMode = 1
        OnMouseClick: execute { iMode := 1; }
    Button (364,353 105x42), "Принять Х1", pressed state: Global_Variables.btnAccept.bX1, invisible if: iMode = 2
        tap Global_Variables.btnAccept.bX1
    Rectangle (115,308 127x30), "%3.2f мм", text variable: curPoint.rPosX0
    Rectangle (115,359 128x30), "%3.2f мм", text variable: curPoint.rPosX1
    Rectangle (115,410 125x30), "%3.2f мм", text variable: curPoint.rPosX2
    Button (228,5 136x40), "Каталог"
        OnMouseDown:  Assign=_Recipe_7inch, Type=Assignment
        OnMouseDown:  ExecuteCommand=ExecuteCommand=[Command=WriteRecipe, Value=sRecGroupName, Value2=sRecName]
        OnMouseDown: execute { bActiveViewRec := TRUE; recipes.getdata(0); }
    Rectangle (109,258 242x30), "%s", text variable: curPoint.name
    Button (364,252 105x42), "Геометрия"
        OnMouseDown:  Dialog=_Diag_geomtry_work, OpenModal=True, PositionX=150, PositionY=50
    Label (10,258 99x30), "Изделие:"
    Image (623,6 36x34), invisible if: NOT Main.bErrLamp, image: Images.Warning
    Button (364,404 105x42), "Принять Х2", pressed state: Global_Variables.btnAccept.bX2, invisible if: iMode = 2
        tap Global_Variables.btnAccept.bX2
    Line (61,115) (431,115)
    Line (61,190) (431,190)
    Label (212,216 317x30), "Точка X0 не установлена", invisible if: NOT Main.fbControl.bNotX0
    Button (481,247 47x47), invisible if: iMode = 2, image: Images.Save
        OnMouseClick: execute {
            IF curPoint.name <> "" AND recipes.screw.name = curPoint.name    THEN
            	recipes.screw := curPoint;
            	recipes.setData(0);
            	recipes.commandRec.ReadRecipe(sRecGroupName,sRecName);
            END_IF
        }
    GroupBox (477,293 313x180), "Актуаторы", invisible if: not SP.bEnAutoMatrix
        Ellipse (53,60 30x30), colour toggle: Actuators.bDr1_enable
        Ellipse (53,60 30x30), invisible if: NOT Actuators.bDr2_error
        Button (12,127 130x45), "Параметры", colour toggle: Main.bErrLamp, invisible if: Actuators.iStage <> 0
            OnMouseDown:  Assign=_Actuators, Type=Assignment
            OnMouseDown: execute { Actuators.bManualMode := TRUE; }
        Label (8,23 33x30), "А1"
        Label (8,60 33x30), "А2"
        Rectangle (106,60 85x30), "%d мм", text variable: Actuators.fbAct2.iCurLength
        Rectangle (106,23 84x30), "%d мм", text variable: Actuators.fbAct1.iCurLength
        Ellipse (53,23 30x30), colour toggle: Actuators.bDr1_enable
        Ellipse (53,23 30x30), invisible if: NOT Actuators.bDr2_error
        Line (198,79) (198,29)
        Button (194,90 100x40), "Пуск", colour toggle: iMode = 2, invisible if: Actuators.iStage <> 0
            tap Actuators.bBtnStart
        Group (7,95 180x30)
            Rectangle (129,0 51x30), "%d", text variable: Actuators.iCycleCnt
            Label (0,0 74x30), "Циклов:"
            Rectangle (74,0 52x30), "%d", text variable: curPoint.iCountCycle
            Label (122,0 13x30), "/"
        Rectangle (212,23 77x30), "%d мм", text variable: Actuators.iCurLenSuport1
        Rectangle (212,60 77x30), "%d мм", text variable: Actuators.iCurLenSuport2
        Line (97,79) (97,29)
        Line (40,79) (40,29)
        Button (194,134 100x40), "Стоп", colour toggle: iMode = 2, invisible if: Actuators.iStage = 0
            tap Actuators.bBtnStop
    Label (199,190 360x30), "Работа актуаторов в цикле", invisible if: Actuators.iStage = 0
END_VISUALIZATION

// Device/Application/Vizualization/7_inch/_Equipment
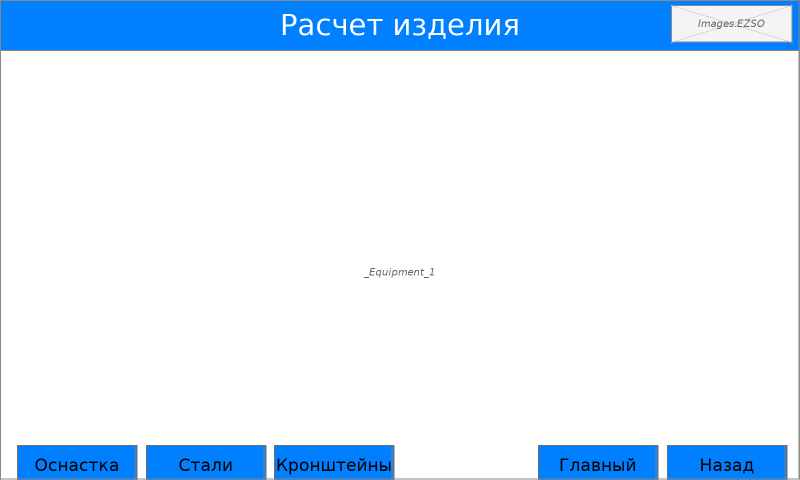
VISUALIZATION _Equipment  // 800x480
    Rectangle (0,0 800x50), "Расчет изделия"
    Image (671,5 121x37), image: Images.EZSO
    TabControl (0,50 800x444)
        shows _Equipment_1()
        shows _Equipment_3()
        shows _Equipment_4()
        shows _Equipment_2()
        [0]: TabTitle=Ввод данных
        [1]: TabTitle=Параметры заготовки
        [2]: TabTitle=Параметры актуаторов, bInvisible=not SP.bEnAutoMatrix
        [3]: TabTitle=Параметры станка
    Button (667,445 120x40), "Назад"
        OnMouseDown:  Assign=_Recipe_7inch, Type=Assignment
    Button (538,445 120x40), "Главный"
        OnMouseDown:  Assign=_MAIN_7inch, Type=Assignment
        OnMouseDown: execute { bActiveViewRec := FALSE; }
    Button (146,445 120x40), "Стали"
        OnMouseDown:  Assign=_Steel_7inch, Type=Assignment
        OnMouseDown: execute { recipes.getdata(2); }
    Button (17,445 120x40), "Оснастка"
        OnMouseDown:  Assign=_Equip_7inch, Type=Assignment
        OnMouseDown: execute { recipes.getdata(1); }
    Button (274,445 120x40), "Кронштейны", invisible if: not SP.bEnAutoMatrix
        OnMouseDown:  Assign=_Support, Type=Assignment
        OnMouseDown: execute { recipes.getdata(3); }
END_VISUALIZATION

// Device/Application/Vizualization/7_inch/_Recipe_7inch
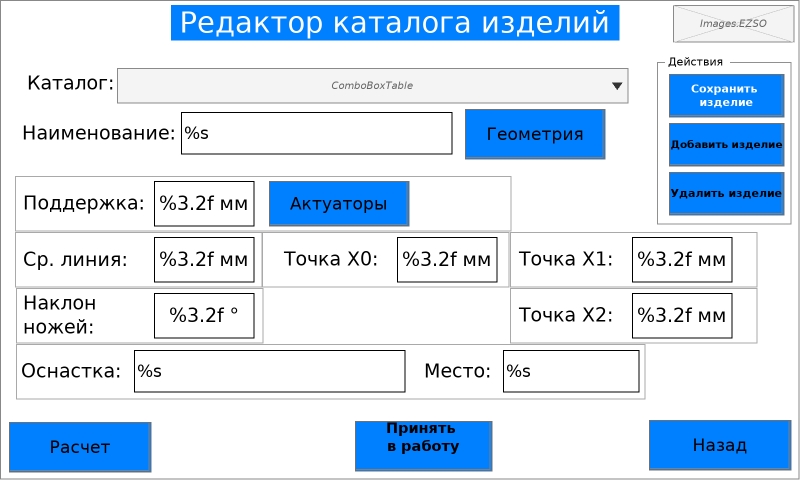
VISUALIZATION _Recipe_7inch  // 800x480, background image Images.background
    RoundedRectangle (15,176 496x55)
    Label (19,118 174x30), "Наименование:"
    Label (24,68 99x30), "Каталог:"
    Image (673,5 121x37), image: Images.EZSO
    Rectangle (171,5 448x35), "Редактор каталога изделий"
    Button (649,420 142x50), "Назад"
        OnMouseDown:  Assign=_MAIN_7inch, Type=Assignment
        OnMouseDown:  ExecuteCommand=ExecuteCommand=[Command=ReadRecipe, Value=sRecGroupName, Value2=sRecName]
        OnMouseDown: execute { bActiveViewRec := FALSE; }
    Button (9,422 142x50), "Расчет"
        OnMouseDown:  Assign=_Equipment, Type=Assignment
        OnMouseDown:  ExecuteCommand=ExecuteCommand=[Command=WriteRecipe, Value=sRecGroupName1, Value2=sRecName1, Command=WriteRecipe, Value=sRecGroupName2, Value2=sRecName2, Command=WriteRecipe, Value=sRecGroupName3, Value2=sRecName3]
    RoundedRectangle (134,350 271x42), "%s", text variable: recipes.Screw.equip.name
        OnMouseDown:  Dialog=_Diag_equip, Parameters={sHeight: , stValue: recipes.Screw.equip.name, sTypeEquip: , sMidle: , sDirection: , sAngle: }, Selected={1: }, OpenModal=True, PositionX=100, PositionY=120
    Label (18,356 106x30), "Оснастка:"
    RoundedRectangle (503,350 136x42), "%s", text variable: recipes.Screw.equip.place
        OnMouseDown: write the text variable via VisuDialogs.Numpad
    Label (421,356 106x30), "Место:"
    GroupBox (657,54 134x170), "Действия"
        Button (12,20 115x43), "Сохранить изделие"
            OnMouseClick: execute { recipes.setData(0); }
        Button (12,118 115x43), "Удалить изделие"
            OnMouseClick: execute { recipes.delData(0); }
        Button (12,69 115x43), "Добавить изделие"
            OnMouseClick: execute { recipes.addData(0); }
    RoundedRectangle (397,237 100x45), "%3.2f мм", text variable: recipes.Screw.rPosX0
        OnMouseClick: write the text variable via VisuDialogs.Numpad, min 0.0, max SP.rMaxLength, title 'Input'
    Label (281,244 105x30), "Точка X0:"
    RoundedRectangle (632,237 100x45), "%3.2f мм", text variable: recipes.Screw.rPosX1
        OnMouseClick: write the text variable via VisuDialogs.Numpad, min 0, max SP.rMaxLength, title 'Input'
    Label (516,244 104x30), "Точка X1:"
    RoundedRectangle (632,293 100x45), "%3.2f мм", text variable: recipes.Screw.rPosX2
        OnMouseClick: write the text variable via VisuDialogs.Numpad, min 0, max SP.rMaxLength, title 'Input'
    Label (516,300 106x30), "Точка X2:"
    Label (20,239 125x41), "Ср. линия:"
    Label (20,186 154x34), "Поддержка:"
    Label (20,294 97x42), "Наклон ножей:"
    RoundedRectangle (181,112 271x42), "%s", text variable: recipes.Screw.name
        OnMouseClick: write the text variable via VisuKbEnRu.Keypad, title 'Input'
    RoundedRectangle (154,181 100x45), "%3.2f мм", text variable: recipes.Screw.rInstal_support
        OnMouseClick: write the text variable via VisuDialogs.Numpad, min 0.0, max 9999, title 'Input'
    RoundedRectangle (154,237 100x45), "%3.2f мм", text variable: recipes.Screw.rMidle_line
        OnMouseClick: write the text variable via VisuDialogs.Numpad, min 0, max 999, title 'Input'
    RoundedRectangle (154,293 100x45), "%3.2f °", text variable: recipes.Screw.rAngle_knives
        OnMouseClick: write the text variable via VisuDialogs.Numpad, min 0, max 999, title 'Input'
    Button (465,109 140x50), "Геометрия"
        OnMouseDown:  Dialog=_Diag_geomtry_rec, OpenModal=True, PositionX=150, PositionY=100
    Button (355,421 137x50), "Принять в работу"
        tap btnAccept.bRec
        OnMouseClick:  Assign=_MAIN_7inch, Type=Assignment
        OnMouseClick:  ExecuteCommand=ExecuteCommand=[Command=ReadRecipe, Value=sRecGroupName, Value2=sRecName]
        OnMouseClick: execute { bActiveViewRec := FALSE; }
    ComboBoxTable (117,68 511x35), variable: recipes.idxArScrew, data array: arScrew
        p1014161805: Global_Variables.SIZE_SCREWS - 0 + 1
        p4234541427: arScrew[INDEX].equip
        p1729500071: arScrew[INDEX].rPosX2
        p286705711: arScrew[INDEX].rPosX1
        p2321883899: arScrew[INDEX].rPosX0
        p4236254150: arScrew[INDEX].rInstal_support
        p1744040210: arScrew[INDEX].rMidle_line
        p290089404: arScrew[INDEX].rAngle_knives
        p2319025000: arScrew[INDEX].rWidth
        p4242324053: arScrew[INDEX].rTurn_step
        p1739542657: arScrew[INDEX].rInner_diam
        p1933151965: ArScrew[INDEX].rOut_diam
        p516019884: arScrew[INDEX].rOut_diam
        p2243050616: arScrew[INDEX].bDirRotate
        p4088588272: arScrew[INDEX].support
        p1757482276: arScrew[INDEX].iActuatorsStartPos
        p505689113: arScrew[INDEX].iActuatorsStep
        p2237128397: arScrew[INDEX].iActuatorsMove
        p4092479075: arScrew[INDEX].iCountCycle
        p1755163831: arScrew[INDEX].rRstmin
        p2232123230: arScrew[INDEX].name
        p511219082: arScrew[INDEX].rRstmax
        OnValueChanged: execute { recipes.getData(0); }
    RoundedRectangle (16,344 629x55)
    RoundedRectangle (15,232 247x55)
    RoundedRectangle (16,288 247x55)
    RoundedRectangle (262,232 247x55)
    RoundedRectangle (510,232 247x55)
    RoundedRectangle (510,288 247x55)
    Button (269,181 140x45), "Актуаторы", invisible if: NOT SP.bEnAutoMatrix
        OnMouseDown:  Dialog=_Diag_support_rec, OpenModal=True, PositionX=150, PositionY=100
END_VISUALIZATION

// Device/Application/Vizualization/7_inch/_Diag_ok
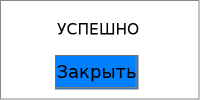
VISUALIZATION _Diag_ok  // 200x100
    Button (55,55 83x34), "Закрыть"
        toggle bGoCalc
        OnMouseClick:  Dialog=Current Dialog, Result=OK, NumpadKeypadSet=True
    Label (43,10 110x38), "УСПЕШНО"
END_VISUALIZATION

// Device/Application/Vizualization/7_inch/_SettingsActuators
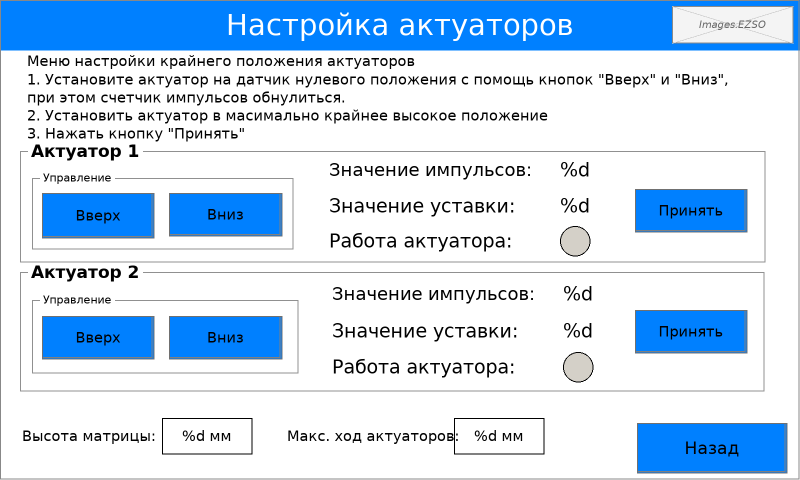
VISUALIZATION _SettingsActuators  // 800x480
    Rectangle (0,0 800x50), "Настройка актуаторов"
    Image (672,6 121x37), image: Images.EZSO
    Button (637,423 150x50), "Назад"
        OnMouseDown:  Assign=_MAIN_7inch, Type=Previous
        OnMouseDown: execute { Actuators.bCalibrateMode :=FALSE; }
    GroupBox (20,143 745x119), "Актуатор 1"
        Label (306,42 206x42), "Значение уставки:"
        Button (615,46 112x43), "Принять", pressed state: Actuators.fbAct1.bCalibrate
            tap Actuators.fbAct1.bCalibrate
        Rectangle (505,48 100x30), "%d", text variable: SP.iMaxImpDr1
        Label (306,7 207x40), "Значение импульсов:"
        Rectangle (505,12 100x30), "%d", text variable: Actuators.iDr1_Cnt
        GroupBox (12,27 261x79), "Управление"
            Button (137,23 113x43), "Вниз", pressed state: Actuators.fbAct1.bBtnBk
                tap Actuators.fbAct1.bBtnBk
            Button (10,23 112x45), "Вверх", pressed state: Actuators.fbAct1.bBtnFrd
                tap Actuators.fbAct1.bBtnFrd
        Ellipse (540,83 30x30), colour toggle: Actuators.bDr1_enable
        Label (306,77 206x42), "Работа актуатора:"
    GroupBox (20,264 744x127), "Актуатор 2"
        GroupBox (12,28 266x81), "Управление"
            Button (10,24 112x43), "Вверх", pressed state: Actuators.fbAct2.bBtnFrd
                tap Actuators.fbAct2.bBtnFrd
            Button (137,24 113x43), "Вниз", pressed state: Actuators.fbAct2.bBtnBk
                tap Actuators.fbAct2.bBtnBk
        Button (615,46 112x43), "Принять", pressed state: Actuators.fbAct2.bCalibrate
            tap Actuators.fbAct2.bCalibrate
        Rectangle (508,52 100x30), "%d", text variable: SP.iMaxImpDr2
        Rectangle (508,15 100x30), "%d", text variable: Actuators.iDr2_Cnt
        Label (309,10 207x40), "Значение импульсов:"
        Label (309,56 206x22), "Значение уставки:"
        Ellipse (543,88 30x30), colour toggle: Actuators.bDr1_enable
        Label (309,82 206x42), "Работа актуатора:"
    Label (24,39 730x117), "Меню настройки крайнего положения актуаторов 1. Установите актуатор на датчик нулевого положения с помощь кнопок "Вверх" и "Вниз", при этом счетчик импульсов обнулиться. 2. Установить актуатор в масимально крайнее высокое положение 3. Нажать кнопку "Принять""
    RoundedRectangle (162,418 90x36), "%d мм", text variable: SP.iHeightMatrix
        OnMouseClick: write the text variable via VisuDialogs.Numpad, min 0, max 1000, title 'Input'
    Label (19,421 141x30), "Высота матрицы:"
    RoundedRectangle (454,418 90x36), "%d мм", text variable: SP.iMaxActuatorsMove
        OnMouseClick: write the text variable via VisuDialogs.Numpad, min 0, max 500, title 'Input'
    Label (284,421 176x30), "Макс. ход актуаторов:"
END_VISUALIZATION

// Device/Application/Vizualization/7_inch/_Diag_equip
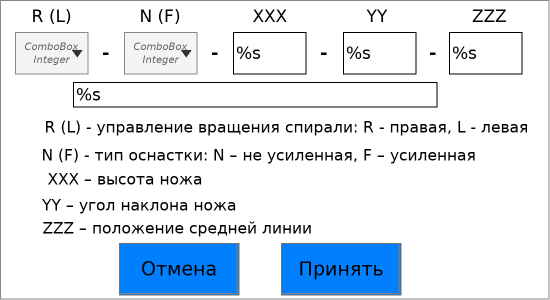
VISUALIZATION _Diag_equip  // 550x300
VAR_IN_OUT
	stValue:WSTRING;	
END_VAR
VAR
	sDirection: INT;
	sTypeEquip:	INT;
	sHeight: WSTRING;
	sAngle:	WSTRING;
	sMidle:	WSTRING;	
END_VAR
    ComboBoxInteger (15,32 73x42), variable: sDirection, text list: 'Direction'
        OnValueChanged: execute {
            stValue := getEquipKeypad(	sDirection,
            	sTypeEquip,
            	sHeight,
            	sAngle,
            	sMidle);
        }
    Label (90,34 32x38), "-"
    ComboBoxInteger (124,32 73x42), variable: sTypeEquip, text list: 'typeEquip'
        OnValueChanged: execute {
            stValue := getEquipKeypad(	sDirection,
            	sTypeEquip,
            	sHeight,
            	sAngle,
            	sMidle);
        }
    Label (199,34 32x38), "-"
    RoundedRectangle (233,32 73x42), "%s", text variable: sHeight
        OnDialogClosed: execute {
            stValue := getEquipKeypad(	sDirection,
            	sTypeEquip,
            	sHeight,
            	sAngle,
            	sMidle);
        }
        OnMouseDown: write the text variable via VisuDialogs.Numpad, min 0, max 999
    Label (308,34 32x38), "-"
    Label (417,34 32x38), "-"
    Label (39,108 495x38), "R (L) - yправление вращения спирали: R - правая, L - левая"
    Label (39,136 440x38), "N (F) - тип оснастки: N – не усиленная, F – усиленная"
    Label (30,-3 49x38), "R (L)"
    Label (137,-3 52x38), "N (F)"
    Label (242,-3 56x38), "XXX"
    Label (361,-3 32x38), "YY"
    Label (463,-3 53x38), "ZZZ"
    Label (39,160 172x38), "XXX – высота ножа"
    Label (39,186 201x38), "YY – угол наклона ножа"
    Label (39,209 277x38), "ZZZ – положение средней линии"
    Button (281,243 120x52), "Принять"
        OnMouseDown:  Dialog=Current Dialog, Result=OK, NumpadKeypadSet=True
    Button (119,243 120x52), "Отмена"
        OnMouseClick:  Dialog=Current Dialog, Result=Cancel, NumpadKeypadSet=True
    RoundedRectangle (73,82 364x25), "%s", text variable: stValue
    RoundedRectangle (343,32 73x42), "%s", text variable: sAngle
        OnDialogClosed: execute {
            stValue := getEquipKeypad(	sDirection,
            	sTypeEquip,
            	sHeight,
            	sAngle,
            	sMidle);
        }
        OnMouseDown: write the text variable via VisuDialogs.Numpad, min 0, max 999
    RoundedRectangle (449,32 73x42), "%s", text variable: sMidle
        OnDialogClosed: execute {
            stValue := getEquipKeypad(	sDirection,
            	sTypeEquip,
            	sHeight,
            	sAngle,
            	sMidle);
        }
        OnMouseDown: write the text variable via VisuDialogs.Numpad, min 0, max 999
END_VISUALIZATION

// Device/Application/Vizualization/7_inch/_SettingsMain_7inch
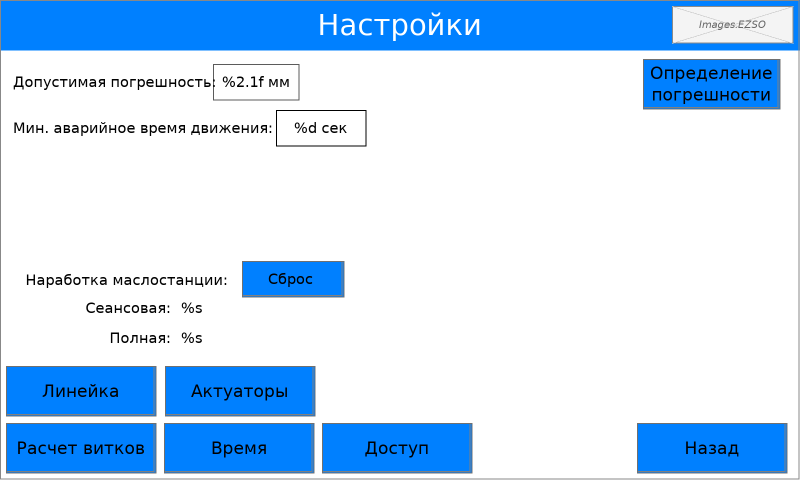
VISUALIZATION _SettingsMain_7inch  // 800x480, background image Images.background1
    Button (637,423 150x50), "Назад"
        OnMouseDown:  Assign=_MAIN_7inch, Type=Assignment
    Button (164,423 150x50), "Время"
        OnMouseDown:  Assign=_TimeSetup_7inch, Type=Assignment
    Button (322,423 150x50), "Доступ"
        OnMouseDown:  Type=OpenUserConfiguration
    Button (242,261 102x36), "Сброс"
        tap bResetOP
    RoundedRectangle (213,64 86x36), "%2.1f мм", text variable: SP.rAccuracy
        OnMouseClick: write the text variable via VisuDialogs.Numpad, min 0, max 9, title 'Input'
    Label (10,67 207x30), "Допустимая погрешность:"
    Button (6,366 150x50), "Линейка"
        OnMouseDown:  Assign=_SettingsSens_7inch, Type=Assignment
    Rectangle (0,0 800x50), "Настройки"
    Rectangle (20,270 211x20), "Наработка маслостанции:"
    Rectangle (32,327 142x22), "Полная:"
    Rectangle (30,297 144x22), "Сеансовая:"
    Rectangle (178,327 123x22), "%s", text variable: Visu_var.stOperTimeTotal
    Rectangle (178,298 121x20), "%s", text variable: Visu_var.stOperTimeSeans
    Image (672,6 121x37), image: Images.EZSO
        OnMouseDown:  Assign=_TypeMachine, Type=Assignment
    RoundedRectangle (276,110 90x36), "%d сек", text variable: SP.iTimeMoveEr
        OnMouseClick: write the text variable via VisuDialogs.Numpad, min 0, max 9999, title 'Input'
    Label (10,113 263x30), "Мин. аварийное время движения:"
    Button (643,59 137x50), "Определение погрешности", colour toggle: iMode = 3
        OnMouseDown: execute { iMode:=3; }
    Button (6,423 150x50), "Расчет витков"
        OnMouseDown:  Assign=_SettingsEquipment, Type=Assignment
    Button (165,366 150x50), "Актуаторы", invisible if: not SP.bEnAutoMatrix
        OnMouseDown:  Assign=_SettingsActuators, Type=Assignment
        OnMouseDown: execute { Actuators.bCalibrateMode := true; }
END_VISUALIZATION

// Device/Application/Vizualization/7_inch/_TimeSetup_7inch
